FUNCTION_BLOCK FB_PunchEngine EXTENDS FB_ComponentBase

VAR PERSISTENT
	nPunchCount					: UDINT;
	fZeroOffset					: LREAL;
END_VAR

VAR	

	// Sequencer
	fbSeq						: FB_Sequence;
	fbSeqOutletBelt				: FB_Sequence;
	
	fVelocity					: LREAL;
	fAcceleration				: LREAL;
	
	fMovePosition				: LREAL;
	bJogPos						: BOOL;
	bJogNeg						: BOOL;
	nPunchRemain				: UINT;
	
	bEnableOutletBelt			: BOOL;
	tIntervallOutletbelt		: TIME;
	tOutletbeltRuntime			: TIME;

	// Watch Variables
	bOutsideMat					: BOOL;
	bPunchDone					: BOOL;
	refObstacle					: REFERENCE TO BOOL;	
	fTravelPosition				: LREAL;
		
	// Parameter
	fPunchHeight				: REAL;
	fPunchHeightAddon			: REAL := 3;
	fPunchVelocity				: LREAL;
	fPunchAcceleration			: LREAL;
	
	// Settings	
	fRodLenght					: REAL;
	fCrankThrow					: REAL;
		
	fMaxVelocity				: LREAL;
	fMinVelocity				: LREAL;
	fDefaultVelocity			: LREAL;
	
	fMaxAcceleration			: LREAL;
	fMinAcceleration			: LREAL;
	fDefaultAcceleration		: LREAL;
	
	fToleranceWindowMM			: LREAL := 0.5;
	fToleranceWindowDeg			: LREAL := 5;
	
	// TorquwLimit
	nTorqueLimit				: INT := 100;
	nTorqueLimitPos				: INT := 100;
	nTorqueLimitNeg				: INT := 10;
		
	// Axis
	bEnable						: BOOL := TRUE;
	refEnable					: REFERENCE TO BOOL;
	fbPunchAxis					: FB_AxisDriver;
	fbOutletbelt				: FB_DigitalOutput;


END_VAR

//TODO: abtransportband!!!!!!

METHOD _Halt : BOOL
VAR_INPUT
END_VAR
fbSeq.Name := 'Halt';

CASE fbSeq.Step OF
	

0	 :	fbSeq.StepDefinition('Punchaxis Halt', T#0S);

		fbPunchAxis.posTorqueLimit := nTorqueLimit;
		fbPunchAxis.negTorqueLimit := nTorqueLimit;
		fbPunchAxis.Halt();		
		fbSeq.NextStep(10);
	
		
10	 :	fbSeq.StepDefinition('', T#0S);
		IF fbPunchAxis.NotMoving THEN
			fbSeq.Finish();
		END_IF
			
END_CASE
END_METHOD

METHOD _Home : BOOL
VAR_INPUT
END_VAR
fbSeq.Name := 'Home';

CASE fbSeq.Step OF
	

0	 :	fbSeq.StepDefinition('Reset Axis', T#0S);

		fbSeq.NextStep(10);
	
	
10	 :	fbSeq.StepDefinition('Set Zero-Position', T#0S);

		fbSeq.NextStep(20);	

		
20	 :	fbSeq.StepDefinition('Move to Zero Postion', T#0S);

		fbSeq.NextStep(30);	

		
30	 :	fbSeq.StepDefinition('', T#0S);

		fbSeq.NextStep(40);

		
40	 :	fbSeq.StepDefinition('', T#0S);

		fbSeq.NextStep(50);

		
50	 :	fbSeq.StepDefinition('', T#0S);

		fbSeq.Finish();

END_CASE
END_METHOD

METHOD _Jog : BOOL
VAR_INPUT
END_VAR
fbSeq.Name := 'Jog';

CASE fbSeq.Step OF
	

0	 :	fbSeq.StepDefinition('Halt Axis', T#0S);
		fbPunchAxis.posTorqueLimit := nTorqueLimit;
		fbPunchAxis.negTorqueLimit := nTorqueLimit;
		fbPunchAxis.Halt();
		fbSeq.NextStep(10);
	
10	 :	fbSeq.StepDefinition('Jog Axis', T#0S);
	
		IF bJogPos OR bJogNeg THEN
			fbPunchAxis.JogAcc(bJogPos , bJogNeg);
		ELSE
			fbSeq.NextStep(20);
		END_IF		
		
20	 :	fbSeq.StepDefinition('Jog Finish', T#0S);
		fbSeq.Finish();

END_CASE
END_METHOD

METHOD _Move : BOOL
VAR
	stMovModParameter			: ST_AxisMoveModParameter;
END_VAR
fbSeq.Name := 'Move';

CASE fbSeq.Step OF
	

0	 :	fbSeq.StepDefinition('Calculate nearest Position', T#0S);
		fbPunchAxis.posTorqueLimit := nTorqueLimit;
		fbPunchAxis.negTorqueLimit := nTorqueLimit;
		
		IF CrankAngle >= 180 THEN
			stMovModParameter.eDirection := MC_Direction.MC_Positive_Direction;
		ELSIF CrankAngle < 180 THEN
			stMovModParameter.eDirection := MC_Direction.MC_Shortest_Way;
		END_IF
		
		stMovModParameter.fPosition := PistonTravelToDeg1(fMovePosition);
		stMovModParameter.fVelocity := fVelocity;
		stMovModParameter.fAcceleration := fAcceleration;
		fbPunchAxis.MoveModEx(stMovModParameter);	
		fbSeq.NextStep(10);
	
	
10	 :	fbSeq.StepDefinition('Position reached', T#0S);
		IF fbPunchAxis.TargetReachedMod(fToleranceWindowDeg) THEN
			fbSeq.Finish();
		END_IF

		
END_CASE
END_METHOD

METHOD _OutletBelt : BOOL
VAR_INPUT
END_VAR
CASE fbSeqOutletBelt.Step OF
	
	0	:	fbSeqOutletBelt.StepDefinition('OutletBelt waiting', T#0S);
			fbSeqOutletBelt.NextStepTransition(10, bEnableOutletBelt);
	
	10	:	fbOutletbelt.SwitchState(TRUE);
			fbSeqOutletBelt.NextStep(20);
			
	20	:	fbSeqOutletBelt.StepDefinition('OutletBelt running', T#0S);
			fbSeqOutletBelt.NextStepDelay(tOutletbeltRuntime, 30);
	
	30	:   fbOutletbelt.SwitchState(FALSE);
			bEnableOutletBelt := FALSE;
			fbSeqOutletBelt.NextStep(40);

	40	:	fbSeqOutletBelt.StepDefinition('OutletBelt resting', T#0S);
			fbSeqOutletBelt.NextStepDelay(tintervallOutletbelt, 0);
	

END_CASE
END_METHOD

METHOD _Punch : BOOL
VAR
	stMovModParameter			: ST_AxisMoveModParameter;
	stMovAddParameter			: ST_AxisMoveAddParameter;
	fPosition					: REAL;
END_VAR
fbSeq.Name := 'Punch';

CASE fbSeq.Step OF
	
0	 :	fbSeq.StepDefinition('Move To Start-Point', T#0S);
		IF fbPunchAxis.TargetReachedMod(fToleranceWindowDeg) THEN
			fbSeq.NextStep(20);
			RETURN;
		END_IF
		
		IF CrankAngle >= 180 THEN
			stMovModParameter.eDirection := MC_Direction.MC_Positive_Direction;
		ELSIF CrankAngle < 180 THEN
			stMovModParameter.eDirection := MC_Direction.MC_Shortest_Way;
		END_IF
		
		fbPunchAxis.posTorqueLimit := nTorqueLimit;
		fbPunchAxis.negTorqueLimit := nTorqueLimit;
				
		stMovModParameter.fPosition := 0;
		stMovModParameter.fVelocity := fDefaultVelocity;
		stMovModParameter.fAcceleration := fDefaultAcceleration;
		stMovModParameter.eBufferMode := MC_BufferMode.MC_Aborting;
		fbPunchAxis.MoveModEx(stMovModParameter);	
		fbSeq.NextStep(10);	
	
10	 :	fbSeq.StepDefinition('Start-Point reached', T#0S);
		IF fbPunchAxis.TargetReachedMod(fToleranceWindowDeg) THEN
			fbSeq.NextStep(20);
		END_IF

20	 :	fbSeq.StepDefinition('Start Punch', T#0S);	
		
		fbPunchAxis.posTorqueLimit := nTorqueLimitPos;
		fbPunchAxis.negTorqueLimit := nTorqueLimitNeg;

		stMovAddParameter.fDistance := 360;
		stMovAddParameter.fVelocity := fPunchVelocity;
		stMovAddParameter.fAcceleration := fPunchAcceleration;
		stMovAddParameter.eBufferMode := MC_BufferMode.MC_Aborting;
		fbPunchAxis.MoveAddEx(stMovAddParameter);	
		fbSeq.NextStep(30);	
		
30	 :	fbSeq.StepDefinition('Punching', T#0S);
		IF InsideMat THEN
			fbSeq.NextStep(40);	
		END_IF			
		
40	 :	fbSeq.StepDefinition('Punching done', T#0S);
		IF OutsideMat THEN
			bPunchDone := TRUE;
			nPunchRemain := nPunchRemain - 1;
			nPunchCount := nPunchCount + 1;
			fbSeq.NextStep(50);	
		END_IF			

50   :	fbSeq.StepDefinition('Check for Continue Punching', T#0S);  
		IF nPunchRemain > 0 THEN
			fbSeq.NextStep(20);	
			RETURN;
		END_IF
		
		fbPunchAxis.posTorqueLimit := nTorqueLimit;
		fbPunchAxis.negTorqueLimit := nTorqueLimit;
			
		IF NOT fbPunchAxis.Moving THEN
			fbSeq.Finish();			
		END_IF	
END_CASE
END_METHOD

/// Actual amplifier temp. [°C]
PROPERTY AmplifierTemp : LREAL
GET
/// Actual amplifier temp. [°C]
AmplifierTemp := fbPunchAxis.AmplifierTemp;
END_GET
END_PROPERTY

PROPERTY BDC : BOOL
GET
BDC := ABS(CrankAngle-180) < fToleranceWindowDeg;
END_GET
END_PROPERTY

PROPERTY CrankAngle : LREAL
GET
VAR
	refAxis				: REFERENCE TO AXIS_REF;
END_VAR
CrankAngle := fbPunchAxis.ActModuloPos;
END_GET
END_PROPERTY

METHOD DegToPistonTravel : LREAL
VAR_INPUT
	fAngle						: LREAL;
END_VAR
VAR
	a							: LREAL;
	b							: LREAL;
	h							: LREAL;
END_VAR
a := fCrankThrow * SIN (DEG_TO_RAD(fAngle));
b := fCrankThrow * COS (DEG_TO_RAD(fAngle));
IF fRodLenght*fRodLenght-a*a < 0 THEN
	RETURN;
END_IF

h := SQRT(fRodLenght*fRodLenght-a*a);

DegToPistonTravel := fCrankThrow - fRodLenght + h - b;


// MANFRED
//a := fCrankThrow * SIN (DEG_TO_RAD(fAngle));
//b := fCrankThrow * COS (DEG_TO_RAD(fAngle));
//
//h1 := fCrankThrow - b;
//h2 := SQRT(fRodLenght*fRodLenght-a*a);
//
//DegToPistonTravel := 2 * fCrankThrow + fRodLenght - h1 - h2;



/// http://www.3d-meier.de/tut16/Kurbel1/Seite1.html	
//DegToPistonTravel := fRodLenght + fCrankThrow - (fCrankThrow * COS(DEG_TO_RAD(fAngle)) + fRodLenght * SQRT(1 - SQRT(fCrankThrow/fRodLenght) * SQRT(SIN(DEG_TO_RAD(fAngle)))));
END_METHOD

METHOD FB_init : BOOL
VAR_INPUT
	bInitRetains : BOOL; // if TRUE, the retain variables are initialized (warm start / cold start)
	bInCopyCode : BOOL;  // if TRUE, the instance afterwards gets moved into the copy code (online change)
END_VAR
eTyp := E_ComponentType.eComponentType_PunchEngine;
END_METHOD

METHOD Halt : E_OperationResult
VAR_INPUT
END_VAR
// init result pessimistic
Halt := E_OperationResult.eOperationResult_NOk;

fbSeq.Start(E_PunchEngineCmd.cmdHalt);

Halt := E_OperationResult.eOperationResult_Ok;
END_METHOD

METHOD Home : E_OperationResult
VAR_INPUT
END_VAR
// init result pessimistic
Home := E_OperationResult.eOperationResult_NOk;

fbSeq.Start(E_PunchEngineCmd.cmdHome);

Home := E_OperationResult.eOperationResult_Ok;
END_METHOD

PROPERTY Homed : BOOL
GET
Homed := fbPunchAxis.Homed;
END_GET
END_PROPERTY

PROPERTY Homing : BOOL
GET
Homing := fbPunchAxis.Homing;
END_GET
END_PROPERTY

PROPERTY InsideMat : BOOL
GET
InsideMat := NOT bOutsideMat;
END_GET
END_PROPERTY

METHOD Jog : E_OperationResult
VAR_INPUT
	JogPos					: BOOL;
	JogNeg					: BOOL;
END_VAR
// init result pessimistic
Jog := E_OperationResult.eOperationResult_NOk;

IF fbSeq.SequenceId <> E_PunchEngineCmd.cmdJog THEN
	fbSeq.Start(E_PunchEngineCmd.cmdJog);
//	RETURN;
END_IF

IF JogPos AND JogNeg THEN
	RETURN;
END_IF

bJogPos := JogPos;
bJogNeg := JogNeg;

Jog := E_OperationResult.eOperationResult_Ok;
END_METHOD

METHOD JogStop : E_OperationResult
// init result pessimistic
JogStop := E_OperationResult.eOperationResult_NOk;

bJogPos := FALSE;
bJogNeg := FALSE;

JogStop := E_OperationResult.eOperationResult_Ok;
END_METHOD

/// Actual motor temp. [°C]
PROPERTY MotorTemp : LREAL
GET
/// Actual motor temp. [°C]
MotorTemp := fbPunchAxis.MotorTemp;
END_GET
END_PROPERTY

METHOD MoveBDC : E_OperationResult
VAR_INPUT
END_VAR
// init result pessimistic
MoveBDC := E_OperationResult.eOperationResult_NOk;

IF ABS(CrankAngle-180) < fToleranceWindowDeg THEN
	RETURN;
END_IF

fMovePosition := 2*fCrankThrow;
fVelocity := fDefaultVelocity; //MAX(MIN(fMaxVelocity, Velocity),fMinVelocity);	
fAcceleration := fDefaultAcceleration;
fbSeq.Start(E_PunchEngineCmd.cmdMove);

MoveBDC := E_OperationResult.eOperationResult_Ok;
END_METHOD

METHOD MovePos : E_OperationResult
VAR_INPUT
	MovePosition			: LREAL;
	Velocity				: LREAL;
END_VAR
// init result pessimistic
MovePos := E_OperationResult.eOperationResult_NOk;

IF ABS(DegToPistonTravel(CrankAngle)-MovePosition) < fToleranceWindowMM THEN
	RETURN;
END_IF

fMovePosition := MovePosition;
fVelocity := MAX(MIN(fMaxVelocity, Velocity),fMinVelocity);	
fAcceleration := fDefaultAcceleration;
fbSeq.Start(E_PunchEngineCmd.cmdMove);

MovePos := E_OperationResult.eOperationResult_Ok;
END_METHOD

METHOD MoveSTART : E_OperationResult
VAR_INPUT
END_VAR
// init result pessimistic
MoveSTART := E_OperationResult.eOperationResult_NOk;

fMovePosition := fCrankThrow*2 - fPunchHeight - fPunchHeightAddon ;
fVelocity := fDefaultVelocity; //MAX(MIN(fMaxVelocity, Velocity),fMinVelocity);	
fAcceleration := fDefaultAcceleration;
fbSeq.Start(E_PunchEngineCmd.cmdMove);

MoveSTART := E_OperationResult.eOperationResult_Ok;
END_METHOD

METHOD MoveTDC : E_OperationResult
VAR_INPUT
END_VAR
// init result pessimistic
MoveTDC := E_OperationResult.eOperationResult_NOk;

IF TDC THEN
	RETURN;
END_IF

fMovePosition := 0;
fVelocity := fDefaultVelocity; //MAX(MIN(fMaxVelocity, Velocity),fMinVelocity);	
fAcceleration := fDefaultAcceleration;
fbSeq.Start(E_PunchEngineCmd.cmdMove);

MoveTDC := E_OperationResult.eOperationResult_Ok;
END_METHOD

PROPERTY Moving : BOOL
GET
Moving := fbPunchAxis.Moving;
END_GET
END_PROPERTY

PROPERTY NotMoving : BOOL
GET
NotMoving := fbPunchAxis.NotMoving;
END_GET
END_PROPERTY

METHOD OutletBeltJog : BOOL
VAR_INPUT
	Enable					: BOOL;
END_VAR
//bEnableOutletBelt := FALSE;
//fbSeqOutletBelt.Init();
IF bEnableOutletBelt THEN
	RETURN;
END_IF
fbOutletbelt.SwitchState(Enable);
END_METHOD

METHOD OutletBeltOnce : BOOL
VAR_INPUT
END_VAR
fbSeqOutletBelt.Init();
tintervallOutletbelt := T#0S;
bEnableOutletBelt := TRUE;
END_METHOD

METHOD OutletBeltSeq : BOOL
VAR_INPUT
	bEnable				: BOOL;
	tIntervall			: UINT;
END_VAR
IF NOT bEnable THEN
	bEnableOutletBelt := FALSE;
	fbSeqOutletBelt.Init();
	fbOutletbelt.SwitchState(FALSE);
ELSE
	bEnableOutletBelt := bEnable;
	tIntervallOutletbelt := DINT_TO_TIME(1000*UINT_TO_DINT(tIntervall));
END_IF
END_METHOD

PROPERTY OutsideMat : BOOL
GET
OutsideMat := bOutsideMat;
END_GET
END_PROPERTY

PROPERTY Override : LREAL
GET
Override := fbPunchAxis.Override;
END_GET
SET
IF Override <> fbPunchAxis.Override THEN
	fbPunchAxis.Override := Override;
	fbPunchAxis.posTorqueLimit := 100;
	fbPunchAxis.negTorqueLimit := 100;
END_IF
END_SET
END_PROPERTY

METHOD PistonTravelToDeg1 : LREAL
VAR_INPUT
	fPistonTravel		: LREAL;
END_VAR
VAR
	h					: LREAL;
	tmp					: LREAL;
END_VAR
IF fPistonTravel > 2 * fCrankThrow OR fPistonTravel < 0 THEN
	RETURN;
END_IF

IF fPistonTravel = 0 THEN
	PistonTravelToDeg1:= 0;	
	RETURN;
END_IF

IF fPistonTravel = 2 * fCrankThrow THEN
	PistonTravelToDeg1:= 180;	
	RETURN;
END_IF

h := fPistonTravel + fRodLenght - fCrankThrow;

tmp := (-fRodLenght*fRodLenght + h*h + fCrankThrow*fCrankThrow)/(2*h*fCrankThrow);

PistonTravelToDeg1:= 180 - rad_to_deg(ACOS(tmp));
END_METHOD

METHOD PistonTravelToDeg2 : LREAL
VAR_INPUT
	fPistonTravel		: LREAL;
END_VAR
VAR
	h					: LREAL;
	tmp					: LREAL;
END_VAR
IF fPistonTravel > 2 * fCrankThrow OR fPistonTravel < 0 THEN
	RETURN;
END_IF

IF fPistonTravel = 0 THEN
	PistonTravelToDeg2:= 0;	
	RETURN;
END_IF

IF fPistonTravel = 2 * fCrankThrow THEN
	PistonTravelToDeg2:= 180;	
	RETURN;
END_IF

h := fPistonTravel + fRodLenght - fCrankThrow;

tmp := (-fRodLenght*fRodLenght + h*h + fCrankThrow*fCrankThrow)/(2*h*fCrankThrow);

PistonTravelToDeg2:= 180 + rad_to_deg(ACOS(tmp));
END_METHOD

METHOD Punch : E_OperationResult
VAR_INPUT
	Continuous				: BOOL;
END_VAR

VAR
	stMovAddParameter			: ST_AxisMoveAddParameter;
END_VAR
// init result pessimistic
Punch := E_OperationResult.eOperationResult_NOk;

fVelocity := MAX(MIN(fMaxVelocity, fPunchVelocity),fMinVelocity);	
fAcceleration := MAX(MIN(fMaxAcceleration, fAcceleration),fMinAcceleration);

bPunchDone:= FALSE;

IF fbseq.SequenceId <> E_PunchEngineCmd.cmdPunch THEN
	nPunchRemain := 1;
	fbSeq.Start(E_PunchEngineCmd.cmdPunch);	
END_IF

IF Continuous THEN
	nPunchRemain := nPunchRemain + 1;
END_IF

Punch := E_OperationResult.eOperationResult_Ok;
END_METHOD

PROPERTY PunchCount : UDINT
GET
PunchCount := nPunchCount;
END_GET
END_PROPERTY

PROPERTY PunchDone : BOOL
GET
PunchDone := bPunchDone;
END_GET
END_PROPERTY

PROPERTY PunchHeight : REAL
GET
PunchHeight := fPunchHeight;
END_GET
SET
fPunchHeight := PunchHeight;
END_SET
END_PROPERTY

PROPERTY Punching : BOOL
GET
Punching := fbSeq.SequenceId = E_PunchEngineCmd.cmdPunch AND fbSeq.State = E_SequenceState.eSequenceState_running;
END_GET
END_PROPERTY

PROPERTY Ready : BOOL
GET
Ready := fbPunchAxis.MotionState <> MC_AXISSTATE_DISABLED;
END_GET
END_PROPERTY

/// Reset component logic
{attribute 'object_name' := 'Reset'}
METHOD Reset
// base logic run
SUPER^.Reset();

fbPunchAxis.Reset();
fbPunchAxis.TorqueLimit := 100;
fbPunchAxis.posTorqueLimit := 100;
fbPunchAxis.negTorqueLimit := 100;

fbOutletbelt.Reset();
nPunchRemain := 0;

fbSeq.Init();			
fbSeqOutletBelt.Init();
END_METHOD

/// Run component logic
{attribute 'object_name' := 'Run'}
METHOD Run : E_ComponentState
// run Base Logic
Run := SUPER^.Run();

IF __ISVALIDREF(refEnable) THEN
	bEnable := refEnable;
END_IF

// run Axis Driver
fbPunchAxis.Run();
fbPunchAxis.Enable := bEnable;
fbPunchAxis.EnablePos := bEnable;
fbPunchAxis.EnableNeg := bEnable;


fbOutletbelt.Run();

// watch Position
fTravelPosition := DegToPistonTravel(CrankAngle);
bOutsideMat := DegToPistonTravel(CrankAngle) < (fCrankThrow*2 - fPunchHeight - fPunchHeightAddon);  

// run Sequences
fbSeq.Enable := TRUE;
fbSeq.Base(FALSE, FALSE);
CASE fbSeq.SequenceId OF	
	E_PunchEngineCmd.cmdMove:	_Move();
	E_PunchEngineCmd.cmdHalt:	_Halt();	
	E_PunchEngineCmd.cmdPunch:	_Punch();	
	E_PunchEngineCmd.cmdHome:	_Home();
	E_PunchEngineCmd.cmdJog:	_Jog();
END_CASE

fbSeqOutletBelt.Enable := TRUE;
fbSeqOutletBelt.Base(FALSE, FALSE);				
_OutletBelt();
END_METHOD

METHOD SetObstacle : BOOL
VAR_IN_OUT
	Obstacle			: BOOL;
END_VAR
refObstacle REF= Obstacle;
END_METHOD

METHOD Setup
VAR_INPUT
	eAxis					: E_Axis;
	eDigitalOutlet			: E_DigitalOutput;
END_VAR
fbPunchAxis.Name := 'Punch Axis';
fbPunchAxis.SetAxisReference(COMP.astAxisRef[eAxis_Punch], COMP.astAxisIO[eAxis_Punch].stIn, COMP.astAxisIO[eAxis_Punch].stOut);
fbPunchAxis.AxisType := E_AxisType.AX5xxx;
fbPunchAxis.DefaultParameter.stMovAbsPrm.fVelocity := 30;
fbPunchAxis.Active := TRUE;
fbPunchAxis.Override := 100;
fbPunchAxis.DefaultParameter.stJogAccPrm.fFastSpeed := 20;
fbPunchAxis.DefaultParameter.stJogAccPrm.fSlowSpeed := 1;
fbPunchAxis.DefaultParameter.stJogAccPrm.tAccTime := T#5S;
fbPunchAxis.EnableLimitSensor:= FALSE;	


fbOutletbelt.Name := 'Outletbelt';
fbOutletbelt.SetReferences(COMP.aStDigitalOutputIO[eDigitalOutput_OutletBelt]);
fbOutletbelt.Active := TRUE;
tOutletbeltRuntime := T#25S;


fMaxVelocity		 := 1111;
fMinVelocity		 := 10;
fDefaultVelocity	 := 180;

fMaxAcceleration	 := 1000000;
fMinAcceleration	 := 0;
fDefaultAcceleration := 0;

fToleranceWindowMM	 := 0.5;
fToleranceWindowDeg	 := 1.5;
END_METHOD

METHOD SetupCrank : BOOL
VAR_INPUT
	fRodLenght				: REAL;
	fCrankThrow				: REAL;
END_VAR
THIS^.fRodLenght	:= fRodLenght;
THIS^.fCrankThrow	:= fCrankThrow;
END_METHOD

METHOD SetupEnable : BOOL

VAR_IN_OUT
	bEnable					: BOOL;
END_VAR
refEnable REF= bEnable;
END_METHOD

METHOD SetupPunch : BOOL
VAR_INPUT
	PunchHeight					: REAL;
	PunchHeightAddon			: REAL;
	MaxVelocity					: LREAL;
	MaxAcceleration				: LREAL;
	TimeBetweenPunch			: LREAL;
END_VAR

VAR
	tmpAngle					: LREAL;
END_VAR
IF TimeBetweenPunch = 0  THEN
	fPunchVelocity := MaxVelocity;
	fPunchAcceleration := MaxAcceleration;
	RETURN;
END_IF

fPunchHeight := PunchHeight;  
fPunchHeightAddon := PunchHeightAddon;


tmpAngle := PistonTravelToDeg1(fCrankThrow*2 - PunchHeight - PunchHeightAddon);

fPunchVelocity := MIN((2*tmpAngle/TimeBetweenPunch), MaxVelocity);
fPunchAcceleration := MaxAcceleration;
END_METHOD

METHOD SetZeroOffset
VAR
	stParam				: st_AxisHomingParameter;
	
END_VAR
fZeroOffset := fbPunchAxis.ActModuloPos;

stParam.fPosition:= 0;
stParam.eHomingMode := MC_HomingMode.MC_Direct; 

fbPunchAxis.HomeEx(stParam);
END_METHOD

PROPERTY TargetReached : BOOL
GET
TargetReached := fbPunchAxis.TargetReachedMod(fToleranceWindowDeg);
END_GET
END_PROPERTY

PROPERTY TDC : BOOL
GET
TDC := ABS(CrankAngle) < fToleranceWindowDeg;
END_GET
END_PROPERTY

/// Actual torque [Nm]
PROPERTY Torque : LREAL
GET
/// Actual torque [Nm]
Torque := fbPunchAxis.Torque;
END_GET
END_PROPERTY

/// The torque limit for both directions. [Nm]
PROPERTY TorqueLimit : INT
GET
/// The torque limit for both directions. [1/10%]
TorqueLimit := nTorqueLimit;
END_GET
SET
nTorqueLimit := TorqueLimit;
END_SET
END_PROPERTY

/// The torque limit for both directions. [Nm]
PROPERTY TorqueLimitNeg : INT
GET
/// The torque limit for both directions. [1/10%]
TorqueLimitNeg := nTorqueLimitNeg;
END_GET
SET
nTorqueLimitNeg := TorqueLimitNeg;
END_SET
END_PROPERTY

/// The torque limit for both directions. [Nm]
PROPERTY TorqueLimitPos : INT
GET
/// The torque limit for both directions. [1/10%]
TorqueLimitPos := nTorqueLimitPos;
END_GET
SET
nTorqueLimitPos := TorqueLimitPos;
END_SET
END_PROPERTY

PROPERTY Velocity : LREAL
GET
Velocity := fVelocity;
END_GET
END_PROPERTY

PROPERTY ZeroOffset : LREAL
GET
ZeroOffset := fZeroOffset;
END_GET
END_PROPERTY

END_FUNCTION_BLOCK

(* stored: Version 1.1.0.1, ProductVersion 3.1.4022.12
   POU FB_PunchEngine: Id {e682466b-149b-46ce-b7ae-08478377e712}, SpecialFunc None
   Folder Commands: Id {d6bb3a00-1415-4c43-b66e-df8e3494eb53}
   Folder Properties: Id {56accc04-24f2-4dea-b365-a22b8d6db586}
   Folder Sequences: Id {b084775c-833a-4b17-883c-4f349cbdff72}
   Folder Setup: Id {e0c74a68-eb11-4486-9516-e8a1d3814c09}
   Folder Utilities: Id {9d7fc255-154d-4fa9-b294-10f7b0134fce}
   Method _Halt: Id {46b7ffab-cde8-4d25-876c-bb43971fd702}
   Method _Home: Id {fb26bee7-3b57-4453-bd61-71ca1b82b4d3}
   Method _Jog: Id {51964e8c-d014-4198-aa12-828738c812d8}
   Method _Move: Id {1625301e-079c-494e-9324-189104430bc6}
   Method _OutletBelt: Id {be91ecec-c9dc-41c9-972e-60484545c7ed}
   Method _Punch: Id {45f639c3-1b9c-49eb-b565-d32ee9a03b04}
   Property AmplifierTemp: Id {66fcad12-d8a9-47ff-a126-33c5aeff7d18}
   Get Get: Id {6a9b1cf2-1b76-491a-8b30-217701ec6d1e}
   Property BDC: Id {c639a29e-3c63-4635-b8e8-d63b2de16559}
   Get Get: Id {eb777667-42be-49bf-956e-0ef2b9509db3}
   Property CrankAngle: Id {210e3655-063d-446d-a518-26d5c639719c}
   Get Get: Id {659526ba-5100-405e-8533-e3cbe4523c43}
   Method DegToPistonTravel: Id {1518b1ad-90a5-4c71-b0d3-517f92c0adf2}
   Method FB_init: Id {6df164eb-9ca2-4370-8952-3273f3d2fb54}
   Method Halt: Id {9500f18b-67be-4594-b414-c1cfd5adde52}
   Method Home: Id {d030df31-c0c2-4ba4-9b1f-ef449cf794cc}
   Property Homed: Id {883803ae-a793-44ab-910f-90856ab6da6d}
   Get Get: Id {ba607391-af9a-4abe-b900-50d73b3c5db8}
   Property Homing: Id {ff6b3481-d658-4509-8e94-8657924d7e39}
   Get Get: Id {e9945973-efcc-46b6-aeb9-3074c448ab78}
   Property InsideMat: Id {0c2fc569-156f-4f3c-9150-26686d1fa485}
   Get Get: Id {fa9bb054-d26a-417b-84e6-88957a8e1725}
   Method Jog: Id {7415a225-522d-41cf-b797-add26ee8988d}
   Method JogStop: Id {8cd0d661-a706-49fc-808b-a8f5b86df139}
   Property MotorTemp: Id {dfc859cc-e9e2-4ef3-98b2-fa61f8f9055e}
   Get Get: Id {85d387e1-487c-40a7-8e03-7bde85830e2c}
   Method MoveBDC: Id {88fb97d9-56d8-4cbb-a0fc-85716abba141}
   Method MovePos: Id {e27ac127-bb4d-485d-9d8c-ae63f363ce97}
   Method MoveSTART: Id {ace88c23-e536-43ef-8cd8-6347db0eaf6d}
   Method MoveTDC: Id {ccba4629-8db2-4b38-8865-6e12cfe60959}
   Property Moving: Id {bfa15079-bda4-44f5-9020-a0fda64195e9}
   Get Get: Id {af174b21-26ab-4fbc-9b8f-61a4516c3353}
   Property NotMoving: Id {bf2c012c-7120-4c7a-9025-b672f8efdd60}
   Get Get: Id {0f56c44c-78bb-49e4-b564-b08686c4b76f}
   Method OutletBeltJog: Id {21617ccf-a8fa-4e63-ab63-b057cc08f188}
   Method OutletBeltOnce: Id {98548120-3b2a-44fe-bcf4-90605d45bc4a}
   Method OutletBeltSeq: Id {3326b6f2-56af-466e-9c33-a51d3a07d217}
   Property OutsideMat: Id {d6c5166c-eb9c-411f-9e4b-06207391dedc}
   Get Get: Id {81f05e00-a2e7-4cbf-856c-f79aafe3bba5}
   Property Override: Id {30a9c1be-4062-4cb7-af1c-d8a6472929fa}
   Get Get: Id {1e8d6658-3a98-4a99-8058-9a85afcd334b}
   Set Set: Id {6f4933c0-9fb5-46d7-81ce-74492a4b6d6c}
   Method PistonTravelToDeg1: Id {bf136d77-3285-47fa-9612-5f9f910d148a}
   Method PistonTravelToDeg2: Id {cb03b3d8-4b16-4193-a913-1a9ca0db5b06}
   Method Punch: Id {5a8a1b3d-f129-4630-8668-1568eb87ed80}
   Property PunchCount: Id {995d008e-30b6-4085-8567-253397661540}
   Get Get: Id {ea4c94ea-7833-4007-9a30-2a356feaa65a}
   Property PunchDone: Id {8e65eb13-4433-496c-9f7c-7f3811424ba1}
   Get Get: Id {84390d25-8fd7-4337-bde4-2ce825d2b69c}
   Property PunchHeight: Id {926984c0-80f2-4705-8585-140bd0aff042}
   Get Get: Id {8eb38317-a13c-450b-af89-908857a117a8}
   Set Set: Id {5ab62919-e283-4f21-8949-e2161c8bbbd3}
   Property Punching: Id {6c7b0d5f-990b-46fb-a1a1-def06d39f8c0}
   Get Get: Id {5229b486-4d14-4f95-9e5d-25202cc7eeeb}
   Property Ready: Id {08ef31d0-3b84-4313-beb1-23b99b15b718}
   Get Get: Id {c8c928ef-612a-4c5d-977d-6aa695ba0e5c}
   Method Reset: Id {cf7a3a72-2e16-46b1-b918-00549dc00d94}
   Method Run: Id {7c75f070-9473-4034-8e74-d30e6747d1e0}
   Method SetObstacle: Id {d5a4d986-d0b8-4a4c-9fa6-45f483c0f9ce}
   Method Setup: Id {f9b5d3bc-fab7-4184-a020-9637294826a2}
   Method SetupCrank: Id {7e7b758d-ba72-459a-ab92-3d38f0f4e896}
   Method SetupEnable: Id {8082b22f-68af-40fc-bbe5-b590738b1112}
   Method SetupPunch: Id {116cd1a8-305b-45f4-91e1-4411a3f332ff}
   Method SetZeroOffset: Id {b297f2b0-c31d-4c8c-a824-50ff9481b738}
   Property TargetReached: Id {e22e93ae-1602-40c8-9b48-ae2edea5157a}
   Get Get: Id {42b47bda-c9ea-46f0-8792-90d0acfef968}
   Property TDC: Id {e3ba09dc-c1e6-4cff-805f-a079aad8bcc7}
   Get Get: Id {48a1f83b-20ba-4a38-8ca0-eb18676e4e1f}
   Property Torque: Id {b39f6def-2c18-4d9b-a159-5077e7a6d690}
   Get Get: Id {04c52b46-a852-4874-9b8a-1f0909b2e22b}
   Property TorqueLimit: Id {c73f6951-37b5-403f-b965-7c7f74721118}
   Get Get: Id {eba28e9a-b239-4262-943a-dd79bd47289e}
   Set Set: Id {b9bad589-cccd-4b9b-91bd-d80c744333d6}
   Property TorqueLimitNeg: Id {db6e1ad0-0d4e-450e-a738-dabae3ce5a06}
   Get Get: Id {5a57e33a-86c1-45a4-b3f2-064eda1cd518}
   Set Set: Id {5b0bdf10-1e3f-4b0d-91e9-d774e01d9b20}
   Property TorqueLimitPos: Id {9de09ef5-d2ad-41d2-ac39-d853e18d0270}
   Get Get: Id {878e451c-d63d-4e5b-bea6-32af84f7a30b}
   Set Set: Id {0ff80f22-1768-4564-b58e-ac1056afe2cd}
   Property Velocity: Id {5d424138-e278-4914-8b83-276943379228}
   Get Get: Id {7bff0bbc-e1b0-4a3c-9fc3-d3d0787040f3}
   Property ZeroOffset: Id {54f4096a-6dd8-4e96-b94c-46f0d3936157}
   Get Get: Id {af92fa33-6cb5-4ac4-9efb-7f265d99dd56} *)
